// TIA Portal V19 export
TYPE "LEXCHANGETRAY_typeRollerIoSignalInterface_B2"
// configuration: LEXCHANGETRAY_typeRollerIoSignalConfigeration_B2
// commands: LEXCHANGETRAY_typeRollerIoSignalManualCommands_B2
// monitoring: LEXCHANGETRAY_typeRollerIoSignalProcessValues_B2
// stored: Access Published
   STRUCT
      configuration : "LEXCHANGETRAY_typeRollerIoSignalConfigeration_B2";
      commands { S7_SetPoint := 'True'} : "LEXCHANGETRAY_typeRollerIoSignalManualCommands_B2";
      monitoring { S7_SetPoint := 'True'} : "LEXCHANGETRAY_typeRollerIoSignalProcessValues_B2";
   END_STRUCT;
END_TYPE
